(* IEC 61131-3 sources: wago_2pump_ebm_fans/PFC200_G2_2ETH_RS_CAN_DPS_T.device.xml.v3^/Plc Logic.plclogic.xml.v3^/Application.application.xml.v3^/BathApp, 7 files *)

(* ---- BATH_APP.fb.st ---- *)
FUNCTION_BLOCK BATH_APP
VAR_INPUT
	Bath :POINTER TO Bath;
END_VAR
VAR
	MainRelayDisable: MR_DISABLE;
	MainRelayEnable: MR_ENABLE;
	FrequenceRecalculate: frequencyCalculate;
	UpdateFanFreq: SET_FREQ_BALANCED;
	CoolingTemp: UINT;
	LiquidAlertTemp: UINT;
	LiquidInTemp: REAL;
	LiquidOutTemp: REAL;
	HighAirTemp: REAL;
	temp_MainStatus: BOOL;
	HA_TC_TOF: TOF;
END_VAR;

LiquidInTemp :=Bath^.LiquidInTemp;
LiquidOutTemp := Bath^.LiquidOutTemp;
HighAirTemp := PV.HighAirTemp;

IF PV.main_remote_command > ENUM_MainStatuses.mainStatusRemoteErrorReset THEN
	IF PV.main_remote_command = ENUM_MainStatuses.mainStatusRemoteSoftShutDown THEN
		Bath^.MainStatus := ENUM_MainStatuses.mainStatusRemoteSoftShutDown;
		MainRelayDisable(Bath := Bath);
		IF LiquidInTemp > Bath^.BathConfig.LiquidTargetTemp -5 OR LiquidOutTemp > Bath^.BathConfig.LiquidTargetTemp -5 THEN
			Bath^.MainKMStatus := TRUE;
			Bath^.PumpKMStatus := TRUE;
			IF Bath^.Freq <> HighAirTemp - 5 THEN
				Bath^.Freq := 100;
				UpdateFanFreq(Bath:= Bath);
			END_IF;
		ELSE
			IF Bath^.Freq <> 0 THEN
				Bath^.Freq := Bath^.BathConfig.FanMinFreq;
				UpdateFanFreq(Bath:= Bath);
			END_IF;
			Bath^.PumpKMStatus := FALSE;
			IF GVL.ContainerAirTemp < HighAirTemp - 5 THEN
				Bath^.MainKMStatus := FALSE;
			ELSE
				Bath^.MainKMStatus := TRUE;
			END_IF;
		END_IF;
	END_IF;

	IF PV.main_remote_command = ENUM_MainStatuses.mainStatusRemoteEmergencyShutDown THEN
		Bath^.MainStatus := ENUM_MainStatuses.mainStatusRemoteEmergencyShutDown;
		MainRelayDisable(Bath := Bath);
		Bath^.PumpKMStatus := FALSE;
		Bath^.MainKMStatus   := FALSE;
		IF Bath^.Freq <> 0 THEN
			Bath^.Freq := Bath^.BathConfig.FanMinFreq;
			UpdateFanFreq(Bath:= Bath);
		END_IF;
	END_IF;

	IF PV.main_remote_command = ENUM_MainStatuses.mainStatusRemoteColdStart THEN
		Bath^.MainStatus := ENUM_MainStatuses.mainStatusRemoteColdStart;
	END_IF;

	IF PV.main_remote_command = ENUM_MAinStatuses.mainStatusRemoteMaintanceMode THEN
		Bath^.MainStatus := ENUM_MAinStatuses.mainStatusRemoteMaintanceMode;
		MainRelayDisable(Bath := Bath);
		Bath^.MainKMStatus := TRUE;
		IF LiquidInTemp > Bath^.BathConfig.LiquidAlertTemp-10 OR LiquidOutTemp > Bath^.BathConfig.LiquidAlertTemp-10 THEN
			Bath^.PumpKMStatus := TRUE;
			IF Bath^.Freq <> 100 THEN
				Bath^.Freq := 100;
				UpdateFanFreq(Bath:= Bath);
			END_IF;
		ELSE
			IF Bath^.Freq <> 0 THEN
				Bath^.Freq := Bath^.BathConfig.FanMinFreq;
				UpdateFanFreq(Bath:= Bath);
			END_IF;
			Bath^.PumpKMStatus := FALSE;
		END_IF;
	END_IF;

	RETURN;
END_IF;

(* Before code only for remote commands *)
IF PV.main_remote_command <= ENUM_MainStatuses.mainStatusRemoteErrorReset AND Bath^.MainStatus >= ENUM_MainStatuses.mainStatusRemoteErrorReset THEN
	Bath^.MainStatus := ENUM_MAinStatuses.statusOK;
END_IF;

IF Bath^.BathConfig.AdminMainRelay =  ENUM_AdminRelayStatus.relayForceDisable THEN
	MainRelayDisable(Bath := Bath);
END_IF
IF GVL.ContainerAirTemp > HighAirTemp THEN
	temp_MainStatus := FALSE;
ELSE
	temp_MainStatus := TRUE;
END_IF;

HA_TC_TOF(IN :=temp_MainStatus, PT := T#5s);
IF  HA_TC_TOF.Q = FALSE THEN
	Bath^.MainStatus := ENUM_MainStatuses.highAirTempStatus;
END_IF;

IF Bath^.MainStatus = ENUM_MainStatuses.statusOK THEN
	//Starting pump
	Bath^.MainKMStatus := TRUE;

	//Checking pressure after pump started
	Bath^.PRESSURE_TC_TON(IN :=Bath^.PumpKMStatus, PT := Bath^.BathConfig.PressureStabilizeInterval);
	IF Bath^.PRESSURE_TC_TON.Q = TRUE THEN
		IF Bath^.PressureOutgoing < Bath^.BathConfig.PressureStabilizeTarget THEN
			Bath^.MainStatus := ENUM_MainStatuses.pressureFail;
		END_IF
	END_IF;

	//Checking Liquid Temperature Sensors
	IF LiquidOutTemp < -50 OR LiquidOuttemp > 200 THEN
		Bath^.TempStatus := ENUM_TempStatuses.tempOutsensorFail;
		Bath^.MainStatus := ENUM_MainStatuses.liquidTempSensorFail;
	END_IF;
	IF LiquidInTemp < -50 OR LiquidIntemp > 200 THEN
		Bath^.TempStatus := ENUM_TempStatuses.tempInsensorFail;
		Bath^.MainStatus := ENUM_MainStatuses.liquidTempSensorFail;
	END_IF;

	IF Bath^.TempStatus = ENUM_TempStatuses.statusOK THEN
		LiquidAlertTemp := Bath^.BathConfig.LiquidAlertTemp;
		//Checking what liquid below Alert temperature
		IF LiquidInTemp > LiquidAlertTemp  THEN
			Bath^.TempStatus := ENUM_TempStatuses.tempLiquidAlert;
			Bath^.MainStatus := ENUM_MainStatuses.highLiquidTempStatus;
		END_IF;
		IF LiquidOutTemp > LiquidAlertTemp THEN
			Bath^.TempStatus := ENUM_TempStatuses.tempLiquidAlert;
			Bath^.MainStatus := ENUM_MainStatuses.highLiquidTempStatus;
		END_IF;
	ELSE
		//If first start or start after error reset, cooling liquid to target
		IF Bath^.TempStatus < ENUM_TempStatuses.tempInSensorFail THEN
			IF LiquidInTemp > Bath^.BathConfig.LiquidTargetTemp  THEN
				Bath^.TempStatus := ENUM_TempStatuses.tempCoolingMode;
				IF Bath^.Freq <> 100 THEN
					Bath^.Freq := 100;
					UpdateFanFreq(Bath:= Bath);
				END_IF;
			ELSE
				IF LiquidInTemp < Bath^.BathConfig.LiquidTargetTemp  THEN
					Bath^.TempStatus := ENUM_TempStatuses.statusOK;
				END_IF;
			END_IF;
		ELSE
			//Checking is sensor connected and working propertly after reseting error
				IF LiquidInTemp > -50 AND LiquidIntemp < 200 THEN
					Bath^.TempStatus := ENUM_TempStatuses.statusOK;
				END_IF;
				IF LiquidOutTemp > -50 AND LiquidOuttemp < 200 THEN
					Bath^.TempStatus := ENUM_TempStatuses.statusOK;
				END_IF;
		END_IF
	END_IF;

	//Cheking level sensor
	IF Bath^.LevelSensor = TRUE THEN
		Bath^.MainStatus := ENUM_MainStatuses.liquidLevelFail;
		Bath^.LevelStatus := ENUM_LevelStatuses.statusFail;
		MainRelayDisable(Bath := Bath);
		Bath^.PumpKMStatus := FALSE;
	ELSE
		Bath^.LevelStatus := ENUM_LevelStatuses.statusOK;
		Bath^.PumpKMStatus := TRUE;
	END_IF;

	//If all ok, working in normal mode
	IF Bath^.LevelStatus = ENUM_LevelStatuses.statusOK
		AND Bath^.TempStatus = ENUM_TempStatuses.statusOK
		AND Bath^.MainStatus = ENUM_MainStatuses.statusOK THEN
		//Timer for fan speed recalculating
		IF Bath^.FanLastReload = FALSE AND Bath^.Bath_Freq_TON.Q = FALSE THEN
			Bath^.FanLastReload := TRUE;
		END_IF
		Bath^.Bath_Freq_TON(IN := Bath^.FanLastReload, PT := Bath^.BathConfig.LiquidStepInterval);
		//Recalculating and setting fan speed
		IF Bath^.Bath_Freq_TON.Q = TRUE THEN
			FrequenceRecalculate(Bath:= Bath);
			UpdateFanFreq(Bath:= Bath);
			Bath^.FanLastReload := FALSE;
		END_IF;

		Bath^.PumpKMStatus := TRUE;
		MainRelayEnable(Bath := Bath);
	END_IF;
ELSE
	IF Bath^.MainStatus <= ENUM_MainStatuses.mainStatusRemoteErrorReset THEN
		MainRelayDisable(Bath := Bath);
	END_IF;
END_IF;

(* ---- BathErrorsFunction.fb.st ---- *)
FUNCTION_BLOCK BathErrorsFunction
VAR_INPUT
END_VAR
VAR_OUTPUT
END_VAR
VAR
	MainRelayDisable: MR_DISABLE;
	MainRelayEnable: MR_ENABLE;
	UpdateFanFreq: SET_FREQ_BALANCED;
	EM_TC_TOF: TOF;

	COLDSTART_TC_TON: TON;
	COLDSTART_PUMP_TC_TON: TON;
	COLDSTART_PUMP_TC_TOF: TOF;

	ColdStartPumpInterval: TIME := T#1s;
	ColdStartPumpCount: UINT := 1;
END_VAR

// Emergency button Press/Unpress
IF GVL.EMERGENCY = TRUE THEN
	GVL.Baths[0].MainKMStatus := FALSE;
	GVL.Baths[1].MainKMStatus := FALSE;
	GVL.Baths[0].PumpKMStatus := FALSE;
	GVL.Baths[1].PumpKMStatus := FALSE;
	MainRelayDisable(Bath := ADR(GVL.Baths[0]));
	MainRelayDisable(Bath := ADR(GVL.Baths[1]));

	GVL.Baths[0].MainStatus := ENUM_MainStatuses.emergencyOn;
	GVL.Baths[1].MainStatus := ENUM_MainStatuses.emergencyOn;
	GVL.Baths[0].Freq := GVL.Baths[0].BathConfig.FanMinFreq;
	GVL.Baths[1].Freq := GVL.Baths[1].BathConfig.FanMinFreq;
END_IF;

IF GVL.Baths[0].MainStatus = ENUM_MainStatuses.emergencyOn OR GVL.Baths[1].MainStatus = ENUM_MainStatuses.emergencyOn THEN
	EM_TC_TOF(IN := GVL.EMERGENCY, PT := T#5S);
	IF  EM_TC_TOF.Q = FALSE THEN
		GVL.Baths[0].MainStatus := ENUM_MainStatuses.statusOK;
		GVL.Baths[1].MainStatus := ENUM_MainStatuses.statusOK;
	END_IF;
END_IF;

// HighAirTemp Inside Container
IF GVL.Baths[0].MainStatus = ENUM_MainStatuses.highAirTempStatus OR GVL.Baths[1].MainStatus = ENUM_MainStatuses.highAirTempStatus THEN
	GVL.Baths[0].MainStatus := ENUM_MainStatuses.highAirTempStatus;
	GVL.Baths[1].MainStatus := ENUM_MainStatuses.highAirTempStatus;
	IF GVL.Baths[0].LiquidInTemp > GVL.Baths[0].BathConfig.LiquidTargetTemp - 5 OR GVL.Baths[1].LiquidInTemp > GVL.Baths[1].BathConfig.LiquidTargetTemp - 5  THEN
		GVL.Baths[0].PumpKMStatus := TRUE;
		GVL.Baths[1].PumpKMStatus := TRUE;
		IF GVL.Baths[0].Freq <> 100 OR GVL.Baths[1].Freq <> 100 THEN
			GVL.Baths[0].Freq := 100;
			GVL.Baths[1].Freq := 100;
			UpdateFanFreq(Bath:= ADR(GVL.Baths[0]));
			UpdateFanFreq(Bath:= ADR(GVL.Baths[1]));
		END_IF;
	ELSE
		GVL.Baths[0].PumpKMStatus := FALSE;
		GVL.Baths[1].PumpKMStatus := FALSE;
		IF GVL.Baths[0].Freq <> 0 OR GVL.Baths[1].Freq <> 0 THEN
			GVL.Baths[0].Freq := GVL.Baths[0].BathConfig.FanMinFreq;
			GVL.Baths[1].Freq := GVL.Baths[1].BathConfig.FanMinFreq;
			UpdateFanFreq(Bath:= ADR(GVL.Baths[0]));
			UpdateFanFreq(Bath:= ADR(GVL.Baths[1]));
		END_IF;
	END_IF;
END_IF;

//High Liquid temp Alert
IF GVL.Baths[0].MainStatus = ENUM_MainStatuses.highLiquidTempStatus OR GVL.Baths[1].MainStatus = ENUM_MainStatuses.highLiquidTempStatus THEN
	IF GVL.Baths[0].MainStatus <> ENUM_MainStatuses.highLiquidTempStatus THEN
		GVL.Baths[0].MainStatus := ENUM_MainStatuses.dependentStatus;
	ELSIF GVL.Baths[1].MainStatus <> ENUM_MainStatuses.highLiquidTempStatus THEN
		GVL.Baths[1].MainStatus := ENUM_MainStatuses.dependentStatus;
	END_IF
	GVL.Baths[0].Freq := GVL.Baths[0].BathConfig.FanMinFreq;
	GVL.Baths[1].Freq := GVL.Baths[1].BathConfig.FanMinFreq;
	UpdateFanFreq(Bath:= ADR(GVL.Baths[0]));
	UpdateFanFreq(Bath:= ADR(GVL.Baths[1]));
	MainRelayDisable(Bath := ADR(GVL.Baths[0]));
	MainRelayDisable(Bath := ADR(GVL.Baths[1]));
	GVL.Baths[0].PumpKMStatus := FALSE;
	GVL.Baths[1].PumpKMStatus := FALSE;
END_IF;

//Pressure Fail temp Alert
IF GVL.Baths[0].MainStatus = ENUM_MainStatuses.pressureFail OR GVL.Baths[1].MainStatus = ENUM_MainStatuses.pressureFail THEN
	IF GVL.Baths[0].MainStatus <> ENUM_MainStatuses.pressureFail THEN
		GVL.Baths[0].MainStatus := ENUM_MainStatuses.dependentStatus;
	ELSIF GVL.Baths[1].MainStatus <> ENUM_MainStatuses.pressureFail THEN
		GVL.Baths[1].MainStatus := ENUM_MainStatuses.dependentStatus;
	END_IF
	GVL.Baths[0].Freq := GVL.Baths[0].BathConfig.FanMinFreq;
	GVL.Baths[1].Freq := GVL.Baths[1].BathConfig.FanMinFreq;
	UpdateFanFreq(Bath:= ADR(GVL.Baths[0]));
	UpdateFanFreq(Bath:= ADR(GVL.Baths[1]));
	MainRelayDisable(Bath := ADR(GVL.Baths[0]));
	MainRelayDisable(Bath := ADR(GVL.Baths[1]));
	GVL.Baths[0].PumpKMStatus := FALSE;
	GVL.Baths[1].PumpKMStatus := FALSE;
END_IF;

//Liquid Level Fail
IF GVL.Baths[0].MainStatus = ENUM_MainStatuses.liquidLevelFail OR GVL.Baths[1].MainStatus = ENUM_MainStatuses.liquidLevelFail THEN
	IF GVL.Baths[0].MainStatus <> ENUM_MainStatuses.liquidLevelFail THEN
		GVL.Baths[0].MainStatus := ENUM_MainStatuses.dependentStatus;
	ELSIF GVL.Baths[1].MainStatus <> ENUM_MainStatuses.liquidLevelFail THEN
		GVL.Baths[1].MainStatus := ENUM_MainStatuses.dependentStatus;
	END_IF
	GVL.Baths[0].Freq := GVL.Baths[0].BathConfig.FanMinFreq;
	GVL.Baths[1].Freq := GVL.Baths[1].BathConfig.FanMinFreq;
	UpdateFanFreq(Bath:= ADR(GVL.Baths[0]));
	UpdateFanFreq(Bath:= ADR(GVL.Baths[1]));
	MainRelayDisable(Bath := ADR(GVL.Baths[0]));
	MainRelayDisable(Bath := ADR(GVL.Baths[1]));
	GVL.Baths[0].PumpKMStatus := FALSE;
	GVL.Baths[1].PumpKMStatus := FALSE;
END_IF;

//Temperature Sensor Fail
IF GVL.Baths[0].MainStatus = ENUM_MainStatuses.liquidTempSensorFail OR GVL.Baths[1].MainStatus = ENUM_MainStatuses.liquidTempSensorFail THEN
	IF GVL.Baths[0].MainStatus <> ENUM_MainStatuses.liquidTempSensorFail THEN
		GVL.Baths[0].MainStatus := ENUM_MainStatuses.dependentStatus;
	ELSIF GVL.Baths[1].MainStatus <> ENUM_MainStatuses.liquidTempSensorFail THEN
		GVL.Baths[1].MainStatus := ENUM_MainStatuses.dependentStatus;
	END_IF
	GVL.Baths[0].Freq := GVL.Baths[0].BathConfig.FanMinFreq;
	GVL.Baths[1].Freq := GVL.Baths[1].BathConfig.FanMinFreq;
	UpdateFanFreq(Bath:= ADR(GVL.Baths[0]));
	UpdateFanFreq(Bath:= ADR(GVL.Baths[1]));
	MainRelayDisable(Bath := ADR(GVL.Baths[0]));
	MainRelayDisable(Bath := ADR(GVL.Baths[1]));
	GVL.Baths[0].PumpKMStatus := FALSE;
	GVL.Baths[1].PumpKMStatus := FALSE;
END_IF;

//ColdStart
IF GVL.Baths[0].MainStatus = ENUM_MainStatuses.mainStatusRemoteColdStart OR GVL.Baths[1].MainStatus = ENUM_MainStatuses.mainStatusRemoteColdStart THEN
	IF ColdStartPumpInterval > T#8S THEN
		PV.main_remote_command := ENUM_MAinStatuses.mainStatusRemoteEmergencyShutDown;
		MainRelayDisable(Bath := ADR(GVL.Baths[0]));
		MainRelayDisable(Bath := ADR(GVL.Baths[1]));
	ELSE
		MainRelayEnable(Bath := ADR(GVL.Baths[0]));
		MainRelayEnable(Bath := ADR(GVL.Baths[1]));
	END_IF

	COLDSTART_TC_TON(IN :=GVL.Baths[0].MainRelayStatus, PT := T#8M);
	IF  COLDSTART_TC_TON.Q = TRUE THEN

		COLDSTART_PUMP_TC_TON(IN :=GVL.Baths[0].PumpKMStatus, PT := ColdStartPumpInterval);
		IF  COLDSTART_PUMP_TC_TON.Q = TRUE THEN
			GVL.Baths[0].PumpKMStatus := FALSE;
			GVL.Baths[1].PumpKMStatus := FALSE;
			IF ColdStartPumpCount = 3 THEN
				ColdStartPumpInterval := ColdStartPumpInterval + T#1S;
				ColdStartPumpCount := 1;
			ELSE
				ColdStartPumpCount := ColdStartPumpCount + 1;
			END_IF
		END_IF;

		COLDSTART_PUMP_TC_TOF(IN :=GVL.Baths[0].PumpKMStatus, PT := T#10S);
		IF  COLDSTART_PUMP_TC_TOF.Q = FALSE THEN
			GVL.Baths[0].PumpKMStatus := TRUE;
			GVL.Baths[1].PumpKMStatus := TRUE;
		END_IF;

	ELSE
		ColdStartPumpInterval := T#1S;
		ColdStartPumpCount := 1;
	END_IF;

END_IF;

// Remote Reset Command
IF PV.main_remote_command = ENUM_MainStatuses.mainStatusRemoteErrorReset THEN
	GVL.Baths[0].MainStatus := ENUM_MAinStatuses.statusOK;
	GVL.Baths[1].MainStatus := ENUM_MAinStatuses.statusOK;
	PV.main_remote_command := 0;
END_IF;

(* ---- frequencyCalculate.fb.st ---- *)
FUNCTION_BLOCK frequencyCalculate
VAR_INPUT
	Bath: POINTER TO Bath;
END_VAR
VAR_OUTPUT
END_VAR
VAR
	freqMax :UINT := 100;
	error, diff1, diff, freqTemp,Kp :REAL;
	LiquidInTemp: REAL;
	LiquidTargetTemp: REAL;
	LiquidDecreaseMax: REAL;
	LiquidIncreaseMax: REAL;
END_VAR

LiquidInTemp := Bath^.LiquidInTemp;
LiquidTargetTemp := Bath^.BathConfig.LiquidTargetTemp;
freqTemp := Bath^.Freq;
LiquidDecreaseMax := Bath^.LiquidDecreaseMax;
LiquidIncreaseMax := Bath^.LiquidIncreaseMax;

IF LiquidInTemp < LiquidDecreaseMax OR LiquidInTemp > LiquidIncreaseMax OR LiquidInTemp > LiquidTargetTemp+2 OR LiquidInTemp < LiquidTargetTemp-2  THEN

	IF LiquidInTemp < LiquidDecreaseMax THEN
		Bath^.LiquidDecreaseMax := LiquidInTemp;
		Bath^.LiquidIncreaseMax := LiquidTargetTemp;
	END_IF;

	IF LiquidInTemp > LiquidIncreaseMax THEN
		Bath^.LiquidIncreaseMax := LiquidInTemp;
		Bath^.LiquidDecreaseMax := LiquidTargetTemp;
	END_IF

	IF LiquidInTemp > LiquidTargetTemp-0.5 OR LiquidInTemp < LiquidTargetTemp+0.5 THEN
		Kp := 1.2;
	ELSE
		Kp := 1;
	END_IF

	error := LiquidInTemp - LiquidTargetTemp;
	diff1 := LiquidTargetTemp / 100 * Kp;
	diff :=diff1 * error;
	freqTemp := freqTemp + diff;

END_IF

IF Bath^.Freq = 0 AND  freqTemp > 0 AND freqTemp < 10 THEN
	freqTemp := 10;
END_IF;

IF freqTemp < Bath^.BathConfig.FanMinFreq THEN
	freqTemp := Bath^.BathConfig.FanMinFreq;
END_IF;

IF freqTemp > freqMax THEN
	freqTemp := freqMax;
END_IF;

Bath^.Freq := freqTemp;

(* ---- MR_DISABLE.fb.st ---- *)
FUNCTION_BLOCK MR_DISABLE
VAR_INPUT
	Bath: POINTER TO Bath;
END_VAR
VAR_OUTPUT
END_VAR
VAR CONSTANT
END_VAR
VAR
	AdminMainRelay: INT;
END_VAR

IF Bath^.MainRelayStatus = TRUE THEN
	AdminMainRelay := Bath^.BathConfig.AdminMainRelay;

	CASE AdminMainRelay OF
		ENUM_AdminRelayStatus.relayForceDisable: Bath^.MainRelay_off := TRUE;
		ENUM_AdminRelayStatus.relayAutoEnable: Bath^.MainRelay_off := TRUE;
		ENUM_AdminRelayStatus.relayForceEnable: Bath^.MainRelay_on := TRUE;
	END_CASE;
END_IF

(* ---- MR_ENABLE.fb.st ---- *)
FUNCTION_BLOCK MR_ENABLE
VAR_INPUT
	Bath: POINTER TO Bath;
END_VAR
VAR_OUTPUT
END_VAR
VAR CONSTANT
END_VAR
VAR
	AdminMainRelay: INT;
END_VAR

IF Bath^.MainRelayStatus = FALSE THEN
	AdminMainRelay := Bath^.BathConfig.AdminMainRelay;

	CASE AdminMainRelay OF
		ENUM_AdminRelayStatus.relayForceDisable: Bath^.MainRelay_off := TRUE;
		ENUM_AdminRelayStatus.relayAutoEnable: Bath^.MainRelay_on := TRUE;
		ENUM_AdminRelayStatus.relayForceEnable: Bath^.MainRelay_on := TRUE;
	END_CASE;
END_IF;

(* ---- SET_FREQ_BALANCED.fb.st ---- *)
FUNCTION_BLOCK SET_FREQ_BALANCED
VAR_INPUT
	Bath: POINTER TO Bath;
END_VAR
VAR_OUTPUT
END_VAR
VAR
	FreqTemp: REAL;
	FanMinVar:WORD := 0;
	FanMaxVar:WORD := 64000;
	Speed:    WORD := 0;
	PW:		  ARRAY[0..5]OF BYTE := [101, 112, 77, 32, 69, 67];
	iCycle:UINT;
END_VAR

FreqTemp := Bath^.Freq;

Speed := REAL_TO_WORD(FanMaxVar / 100 * FreqTemp);

IF Speed < FanMinVar THEN
	Speed := FanMinVar;
END_IF;
IF Speed > FanMaxVar THEN
	Speed := FanMaxVar;
END_IF;

FOR iCycle := 1 TO 12 BY 1 DO
	Bath^.Fans[iCycle].Speed := Speed;
END_FOR;

(* ---- BATH_PRG.prg.st ---- *)
PROGRAM BATH_PRG
VAR
	iCycle: UINT;
	App: BATH_APP;
	START 	:BOOL := FALSE;
	BathErrorsFunction: BathErrorsFunction;
END_VAR

IF START = FALSE THEN
	START := TRUE;
	GVL.Baths[0].BathConfig := PV.BathConfigs[0];
	GVL.Baths[1].BathConfig := PV.BathConfigs[1];
END_IF

IF (GVL.QFUndervoltage = FALSE) THEN
	GVL.QFUndervoltage := TRUE;
ELSE
	App(Bath:= ADR(GVL.Baths[0]));
	App(Bath:= ADR(GVL.Baths[1]));

	BathErrorsFunction();
END_IF
